(*

## Short summary
This class provides assert statements for UTF-8 strings up to 255 bytes length

**Attention:** 
	All strings are handled as null-terminated byte streams

.. <legal notes>

legal notes
=================
| SPDX-FileCopyrightText: © 2024 ekvip automation GmbH <info@ekvip.de>
| SPDX-License-Identifier: Apache-2.0
| For details check: Apache-2.0_

.. _Apache-2.0: https://www.apache.org/licenses/LICENSE-2.0

.. </legal notes>



*)

{attribute 'reflection'}
FUNCTION_BLOCK INTERNAL Utf8StringAssertions EXTENDS AbstractAssertion IMPLEMENTS IUtf8StringAssertions
VAR
	(* class to handle the UTF-8 string assertions *)  
	assertion	:Utf8StringPointerAssertions();
END_VAR

(*

## Short summary
This abstract property returns the class name of the concrete object, 
It's for debugging purpose

.. <legal notes>

legal notes
=================
| SPDX-FileCopyrightText: © 2022 ekvip automation GmbH <info@ekvip.de>
| SPDX-License-Identifier: Apache-2.0
| For details check: Apache-2.0_

.. _Apache-2.0: https://www.apache.org/licenses/LICENSE-2.0

.. </legal notes>

*)

PROPERTY className :CNM_AbstractObject.ClassName
GET
className := 'CNM_Assertor.Utf8StringAssertions';
END_GET
END_PROPERTY

(*

## Short summary
This assertion method checks if the current string ``stringToCheck`` contains the search string ``searchString``.
Processed strings must be in UTF-8 encoding

.. <legal notes>

legal notes
=================
| SPDX-FileCopyrightText: © 2024 ekvip automation GmbH <info@ekvip.de>
| SPDX-License-Identifier: Apache-2.0
| For details check: Apache-2.0_

.. _Apache-2.0: https://www.apache.org/licenses/LICENSE-2.0

.. </legal notes>



*)

METHOD contains
VAR_INPUT
	(* current string to check *)
	{attribute 'TcEncoding' := 'UTF-8'}
	stringToCheck	:Tc2_System.T_MaxString;
	(* string must be found in ``stringToCheck`` *)
	{attribute 'TcEncoding' := 'UTF-8'}
	searchString	:Tc2_System.T_MaxString;
	(* message if the assertion is false *)
	message			:AssertMessage;
	(* ``TRUE`` means ignore cases; ``FALSE`` means that cases must be equal too *)
	ignoreCases		:BOOL := FALSE;
	(*normalize both strings for check*)
	normalizeStrings :BOOL := TRUE;
END_VAR
assertion.contains(
	stringToCheck 	:= ADR(stringToCheck),
	searchString  	:= ADR(searchString),
	ignoreCases 	:= ignoreCases,
	message 		:= message,
	normalizeStrings := normalizeStrings
);
END_METHOD

(*

## Short summary
This assertion method checks if the current string ``stringToCheck`` doesn't contain the search string ``searchString``.
Processed strings must be in UTF-8 encoding

.. <legal notes>

legal notes
=================
| SPDX-FileCopyrightText: © 2024 ekvip automation GmbH <info@ekvip.de>
| SPDX-License-Identifier: Apache-2.0
| For details check: Apache-2.0_

.. _Apache-2.0: https://www.apache.org/licenses/LICENSE-2.0

.. </legal notes>



*)

METHOD containsNo
VAR_INPUT
	(* current string to check *)
	{attribute 'TcEncoding' := 'UTF-8'}
	stringToCheck	:Tc2_System.T_MaxString;
	(* string that must not be found in ``stringToCheck`` *)
	{attribute 'TcEncoding' := 'UTF-8'}
	searchString	:Tc2_System.T_MaxString;
	(* message if the assertion is false *)
	message			:AssertMessage;
	(* ``TRUE`` means ignore cases; ``FALSE`` means that cases must be equal too *)
	ignoreCases		:BOOL := FALSE;
	(*normalize both strings for check*)
	normalizeStrings :BOOL := TRUE;
END_VAR
THIS^.assertion.containsNo(
	stringToCheck 	:= ADR(stringToCheck),
	searchString  	:= ADR(searchString),
	ignoreCases 	:= ignoreCases,
	message 		:= message,
	normalizeStrings := normalizeStrings
);
END_METHOD

(*

## Short summary
This assertion method checks if the current string ``stringToCheck`` ends with the string ``end``.
Processed strings must be in UTF-8 encoding

.. <legal notes>

legal notes
=================
| SPDX-FileCopyrightText: © 2024 ekvip automation GmbH <info@ekvip.de>
| SPDX-License-Identifier: Apache-2.0
| For details check: Apache-2.0_

.. _Apache-2.0: https://www.apache.org/licenses/LICENSE-2.0

.. </legal notes>



*)

METHOD endsWith
VAR_INPUT
	(* current string to check *)
	{attribute 'TcEncoding' := 'UTF-8'}
	stringToCheck	:Tc2_System.T_MaxString;
	(* expected end of ``stringToCheck`` *)
	{attribute 'TcEncoding' := 'UTF-8'}
	end				:Tc2_System.T_MaxString;
	(* message if the assertion is false *)
	message			:AssertMessage;
	(* ``TRUE`` means ignore cases; ``FALSE`` means that cases must be equal too *)
	ignoreCases		:BOOL := FALSE;
	(* ``TRUE`` means truncation of spaces on the right side of ``stringToCheck``*)
	trim		:BOOL := FALSE;
	(*normalize both strings for check*)
	normalizeStrings :BOOL := TRUE;
END_VAR
assertion.endsWith(
	stringToCheck	:= ADR(stringToCheck),
	end				:= ADR(end),
	ignoreCases		:= ignoreCases,
	trim		:= trim,
	message			:= message,
	normalizeStrings := normalizeStrings
);
END_METHOD

(*

## Short summary
This assertion method checks if the current string ``stringToCheck`` is empty.
Processed strings must be in UTF-8 encoding

.. <legal notes>

legal notes
=================
| SPDX-FileCopyrightText: © 2024 ekvip automation GmbH <info@ekvip.de>
| SPDX-License-Identifier: Apache-2.0
| For details check: Apache-2.0_

.. _Apache-2.0: https://www.apache.org/licenses/LICENSE-2.0

.. </legal notes>



*)

METHOD isEmpty
VAR_INPUT
	(* current string to check *)
	{attribute 'TcEncoding' := 'UTF-8'}
	stringToCheck	:Tc2_System.T_MaxString;
	(* message if the assertion is false *)
	message			:AssertMessage;
END_VAR
IF (stringToCheck <> '') THEN
	THIS^.assertionWasWrong(message, THIS^.getDebugInfo('isEmpty'));
END_IF
END_METHOD

(*

## Short summary
This assertion method checks if the current string ``stringToCheck`` is equal to ``expected``.
Processed strings must be in UTF-8 encoding

.. <legal notes>

legal notes
=================
| SPDX-FileCopyrightText: © 2024 ekvip automation GmbH <info@ekvip.de>
| SPDX-License-Identifier: Apache-2.0
| For details check: Apache-2.0_

.. _Apache-2.0: https://www.apache.org/licenses/LICENSE-2.0

.. </legal notes>



*)

METHOD isEqualTo
VAR_INPUT
	(* current string to check *)
	{attribute 'TcEncoding' := 'UTF-8'}
	stringToCheck	:Tc2_System.T_MaxString;
	(* ``stringToCheck`` must be equal to expected *)
	{attribute 'TcEncoding' := 'UTF-8'}
	expected		:Tc2_System.T_MaxString;
	(* message if the assertion is false *)
	message			:AssertMessage;
	(* ``TRUE`` means ignore cases; ``FALSE`` means that cases must be equal too *)
	ignoreCases		:BOOL := FALSE;
	(*normalize both strings for check*)
	normalizeStrings :BOOL := TRUE;
END_VAR
assertion.isEqualTo(
	stringToCheck	:= ADR(stringToCheck),
	expected		:= ADR(expected),
	ignoreCases		:= ignoreCases,
	message			:= message,
	normalizeStrings := normalizeStrings
);
END_METHOD

(*

## Short summary
This assertion method checks if the current string ``stringToCheck`` is not empty.
Processed strings must be in UTF-8 encoding

.. <legal notes>

legal notes
=================
| SPDX-FileCopyrightText: © 2024 ekvip automation GmbH <info@ekvip.de>
| SPDX-License-Identifier: Apache-2.0
| For details check: Apache-2.0_

.. _Apache-2.0: https://www.apache.org/licenses/LICENSE-2.0

.. </legal notes>



*)

METHOD isNotEmpty
VAR_INPUT
	(* current string to check *)
	{attribute 'TcEncoding' := 'UTF-8'}
	stringToCheck	:Tc2_System.T_MaxString;
	(* message if the assertion is false *)
	message			:AssertMessage;
END_VAR
IF (stringToCheck = '') THEN
	THIS^.assertionWasWrong(message, THIS^.getDebugInfo('isEmpty'));
END_IF
END_METHOD

(*

## Short summary
This assertion method checks if the current string ``stringToCheck`` is not equal to ``unexpected``.
Processed strings must be in UTF-8 encoding

.. <legal notes>

legal notes
=================
| SPDX-FileCopyrightText: © 2024 ekvip automation GmbH <info@ekvip.de>
| SPDX-License-Identifier: Apache-2.0
| For details check: Apache-2.0_

.. _Apache-2.0: https://www.apache.org/licenses/LICENSE-2.0

.. </legal notes>



*)

METHOD isNotEqualTo
VAR_INPUT
	(* current string to check *)
	{attribute 'TcEncoding' := 'UTF-8'}
	stringToCheck	:Tc2_System.T_MaxString;
	(* ``stringToCheck`` must be not equal to expected *)
	{attribute 'TcEncoding' := 'UTF-8'}
	unexpected		:Tc2_System.T_MaxString;
	(* message if the assertion is false *)
	message			:AssertMessage;
	(* ``TRUE`` means ignore cases; ``FALSE`` means that cases must be equal too *)
	ignoreCases		:BOOL := FALSE;
	(*normalize both strings for check*)
	normalizeStrings :BOOL := TRUE;
END_VAR
THIS^.assertion.isNotEqualTo(
	stringToCheck	:= ADR(stringToCheck),
	unexpected		:= ADR(unexpected),
	ignoreCases		:= ignoreCases,
	message			:= message,
	normalizeStrings := normalizeStrings
);
END_METHOD

(*

## Short summary
This assertion method checks if the current string ``stringToCheck`` length is between ``minLength`` and ``maxLength``.
Processed strings must be in UTF-8 encoding

.. <legal notes>

legal notes
=================
| SPDX-FileCopyrightText: © 2024 ekvip automation GmbH <info@ekvip.de>
| SPDX-License-Identifier: Apache-2.0
| For details check: Apache-2.0_

.. _Apache-2.0: https://www.apache.org/licenses/LICENSE-2.0

.. </legal notes>



*)

METHOD lengthIsBetween
VAR_INPUT
	(* current string to check *)
	{attribute 'TcEncoding' := 'UTF-8'}
	stringToCheck		:Tc2_System.T_MaxString;
	(* lower limit of the string length *)
	minLength			:USINT;
	(* upper limit of the string length *)
	maxLength			:USINT;
	(* string length units of measurement *)
	stringLengthUnit	:UnicodeStringLengthUnit;
	(* message if the assertion is false *)
	message				:AssertMessage;
END_VAR
THIS^.assertion.lengthIsBetween(
	stringToCheck		:= ADR(stringToCheck),
	minLength			:= minLength,
	maxLength			:= maxLength,
	stringLengthUnit	:= stringLengthUnit,
	message				:= message
);
END_METHOD

(*

## Short summary
This assertion method checks if the current string ``stringToCheck`` length is equal to ``expectedLength``.
Processed strings must be in UTF-8 encoding

.. <legal notes>

legal notes
=================
| SPDX-FileCopyrightText: © 2024 ekvip automation GmbH <info@ekvip.de>
| SPDX-License-Identifier: Apache-2.0
| For details check: Apache-2.0_

.. _Apache-2.0: https://www.apache.org/licenses/LICENSE-2.0

.. </legal notes>



*)

METHOD lengthIsExact
VAR_INPUT
	(* current string to check *)
	{attribute 'TcEncoding' := 'UTF-8'}
	stringToCheck		:Tc2_System.T_MaxString;
	(* expected length of ``stringToCheck`` *)
	expectedLength		:USINT;
	(* string length units of measurement *)
	stringLengthUnit	:UnicodeStringLengthUnit;
	(* message if the assertion is false *)
	message				:AssertMessage;
END_VAR
THIS^.assertion.lengthIsExact(
	stringToCheck		:= ADR(stringToCheck),
	expectedLength		:= expectedLength,
	stringLengthUnit	:= stringLengthUnit,
	message				:= message
);
END_METHOD

(*

## Short summary
This assertion method checks if the current string ``stringToCheck`` length is equal or less than to ``maxLength``.
Processed strings must be in UTF-8 encoding

.. <legal notes>

legal notes
=================
| SPDX-FileCopyrightText: © 2024 ekvip automation GmbH <info@ekvip.de>
| SPDX-License-Identifier: Apache-2.0
| For details check: Apache-2.0_

.. _Apache-2.0: https://www.apache.org/licenses/LICENSE-2.0

.. </legal notes>



*)

METHOD lengthIsMax
VAR_INPUT
	(* current string to check *)
	{attribute 'TcEncoding' := 'UTF-8'}
	stringToCheck		:Tc2_System.T_MaxString;
	(* upper limit of the length of ``stringToCheck`` *)
	maxLength			:USINT;
	(* string length units of measurement *)
	stringLengthUnit	:UnicodeStringLengthUnit;
	(* message if the assertion is false *)
	message				:AssertMessage;
END_VAR
THIS^.assertion.lengthIsMax(
	stringToCheck		:= ADR(stringToCheck),
	maxLength			:= maxLength,
	stringLengthUnit	:= stringLengthUnit,
	message				:= message
);
END_METHOD

(*

## Short summary
This assertion method checks if the current string ``stringToCheck`` length is equal or greater than to ``minLength``.
Processed strings must be in UTF-8 encoding

.. <legal notes>

legal notes
=================
| SPDX-FileCopyrightText: © 2024 ekvip automation GmbH <info@ekvip.de>
| SPDX-License-Identifier: Apache-2.0
| For details check: Apache-2.0_

.. _Apache-2.0: https://www.apache.org/licenses/LICENSE-2.0

.. </legal notes>



*)

METHOD lengthIsMin
VAR_INPUT
	(* current string to check *)
	{attribute 'TcEncoding' := 'UTF-8'}
	stringToCheck		:Tc2_System.T_MaxString;
	(* lower limit of the length of ``stringToCheck`` *)
	minLength			:USINT;
	(* string length units of measurement *)
	stringLengthUnit	:UnicodeStringLengthUnit;
	(* message if the assertion is false *)
	message				:AssertMessage;
END_VAR
THIS^.assertion.lengthIsMin(
	stringToCheck		:= ADR(stringToCheck),
	minLength			:= minLength,
	stringLengthUnit	:= stringLengthUnit,
	message				:= message
);
END_METHOD

(*

## Short summary
This methods is the setter for the callback class if an assertion was false

.. <legal notes>

legal notes
=================
| SPDX-FileCopyrightText: © 2024 ekvip automation GmbH <info@ekvip.de>
| SPDX-License-Identifier: Apache-2.0
| For details check: Apache-2.0_

.. _Apache-2.0: https://www.apache.org/licenses/LICENSE-2.0

.. </legal notes>



*)

METHOD setCallBack
VAR_INPUT
	(* the class that must be informed if an assertion is false *)
	callBack	:IAssertCallBack;  
END_VAR
SUPER^.setCallBack(callBack);
THIS^.assertion.setCallBack(callBack);
END_METHOD

(*

## Short summary
This assertion method checks if the current string ``stringToCheck`` starts with string ``start``.
Processed strings must be in UTF-8 encoding

.. <legal notes>

legal notes
=================
| SPDX-FileCopyrightText: © 2024 ekvip automation GmbH <info@ekvip.de>
| SPDX-License-Identifier: Apache-2.0
| For details check: Apache-2.0_

.. _Apache-2.0: https://www.apache.org/licenses/LICENSE-2.0

.. </legal notes>



*)

METHOD startsWith
VAR_INPUT
	(* current string to check *)
	{attribute 'TcEncoding' := 'UTF-8'}
	stringToCheck	:Tc2_System.T_MaxString;
	(* expected start of ``stringToCheck`` *)
	{attribute 'TcEncoding' := 'UTF-8'}
	start			:Tc2_System.T_MaxString;
	(* message if the assertion is false *)
	message			:AssertMessage;
	(* ``TRUE`` means ignore cases; ``FALSE`` means that cases must be equal too *)
	ignoreCases		:BOOL := FALSE;
	(* ``TRUE`` means truncation of spaces on the left side of ``stringToCheck``*)
	trim		:BOOL := FALSE;
	(*normalize both strings for check*)
	normalizeStrings :BOOL := TRUE;
END_VAR
assertion.startsWith(
	stringToCheck	:= ADR(stringToCheck),
	start			:= ADR(start),
	ignoreCases		:= ignoreCases,
	trim		:= trim,
	message			:= message,
	normalizeStrings := normalizeStrings
);
END_METHOD

END_FUNCTION_BLOCK

(* stored: Version 1.1.0.1, ProductVersion 3.1.4026.12
   POU Utf8StringAssertions: Id {a41418c7-5c67-49f1-96bd-7ca608dfb3ff}, SpecialFunc None
   Property className: Id {c47f3da8-3028-428c-99dc-152561a16a4b}
   Get Get: Id {fd9932fc-f2f1-48f2-83ef-36ef368255fa}
   Method contains: Id {958f0556-bc07-45a2-a21b-fdd4d30b9483}
   Method containsNo: Id {d35575f5-4dce-4228-bc74-9fcddd791faf}
   Method endsWith: Id {18c96a67-fb27-4e96-ad14-bed15424351c}
   Method isEmpty: Id {c9b836ee-b7c0-4854-ab7d-6618a010c133}
   Method isEqualTo: Id {b835eb13-17cd-4cbe-bd33-831e8efc6d28}
   Method isNotEmpty: Id {d1512cba-e22a-44b1-8a64-0806ef5301e9}
   Method isNotEqualTo: Id {e6dac070-0ce3-494f-8740-3b7c6120c64e}
   Method lengthIsBetween: Id {7f4e89c9-1950-43d5-8e05-58078c012d4a}
   Method lengthIsExact: Id {0b4a8869-dcca-4b91-beb7-3c038385685a}
   Method lengthIsMax: Id {8fb9f4cc-b224-416d-a102-6077f70b72ef}
   Method lengthIsMin: Id {64e93fec-98d2-4cbd-9c6c-2ce783224e9c}
   Method setCallBack: Id {0d3cb4ee-41cb-4009-9e03-0ec5170e70c5}
   Method startsWith: Id {912b665f-6499-4931-86dc-e5138446d9f2} *)
